PROGRAM IO
VAR


	Scaled_control: LREAL;

END_VAR


	

GVL.Temp := 0.010071*INT_TO_LREAL(GVL.tempSensor) - 39.996;//((INT_TO_LREAL(GVL.tempSensor)/3.2767) - 0.2424*5000)*165/5000; //Scaled for 0-5V with range -20 to 70C. See documentation for sensor
GVL.Humidity := (INT_TO_LREAL(IO_VARS.HUM_SENS)/3.2767)*100/5000;



IF GVL.manualMode=FALSE THEN
	
////////////MAPPING METAL HALIDE LIGHTS/////////////
IF GVL.Light1Level=0 THEN
	IO_VARS.MH1:=0;
	IO_VARS.MH2:=0;
	IO_VARS.MH3:=0;
ELSIF  GVL.Light1Level=1 THEN
	IO_VARS.MH1:=1;
	IO_VARS.MH2:=0;
	IO_VARS.MH3:=0;
ELSIF  GVL.Light1Level=2 THEN
	IO_VARS.MH1:=1;
	IO_VARS.MH2:=1;
	IO_VARS.MH3:=0;
ELSIF  GVL.Light1Level=3 THEN
	IO_VARS.MH1:=1;
	IO_VARS.MH2:=1;
	IO_VARS.MH3:=1;
END_IF

////////////MAPPING HIGH PRESSURE SODIUM LIGHTS/////////////
IF GVL.Light2Level=0 THEN
	IO_VARS.HPS1:=0;
	IO_VARS.HPS2:=0;
	IO_VARS.HPS3:=0;
ELSIF  GVL.Light2Level=1 THEN
	IO_VARS.HPS1:=1;
	IO_VARS.HPS2:=0;
	IO_VARS.HPS3:=0;
ELSIF  GVL.Light2Level=2 THEN
	IO_VARS.HPS1:=1;
	IO_VARS.HPS2:=1;
	IO_VARS.HPS3:=0;
ELSIF  GVL.Light2Level=3 THEN
	IO_VARS.HPS1:=1;
	IO_VARS.HPS2:=1;
	IO_VARS.HPS3:=1;
END_IF
	
END_IF

END_PROGRAM

(* stored: Version 1.1.0.1, ProductVersion 3.1.4022.18
   POU IO: Id {1ce9b422-5f87-4557-abb2-cabcfdf99a7f}, SpecialFunc None *)
